// TIA Portal project "Project1" (V15)

(* hardware
DEVICE "PC-System_1"  SIMATIC PC station
   slot 0: "SIMATIC PC station"  Rail  SIMATIC PC-Station  V1.0
      slot 125: "Stationmanager"  Station_Manager  V6.0.4
   slot 1: "HMI_RT_1"  WinCC RT Professional  6AV2 105-0xxxx-xxxx  15.0.0.0
   slot 2: "IE general_1"  IE General  IE_CP  V8.2.0
DEVICE "S7-1200 station_1"  S7-1200 Station
   slot 0: "Rack_0"  S7-1200 Rack  Rack  V1.0
   slot 1: "PLC_1"  CPU 1212C DC/DC/DC  6ES7 212-1AE40-0XB0  V4.2
*)

// ===== PLC "PLC_1"  CPU 1212C DC/DC/DC =====

VAR_GLOBAL   // PLC tag table "Default tag table"
   "In1" AT %M0.0 : Bool;
   "Out1" AT %M0.1 : Bool;
END_VAR

ORGANIZATION_BLOCK "Main"   // OB1, LAD, ProgramCycle
TITLE = "Main Program Sweep (Cycle)"
{ S7_Optimized_Access := 'TRUE' }
VERSION : 0.1
   VAR_INPUT
      Initial_Call : Bool;   // Initial call of this OB
      Remanence : Bool;   // =True, if remanent data are available
   END_VAR
BEGIN

REGION Network 1
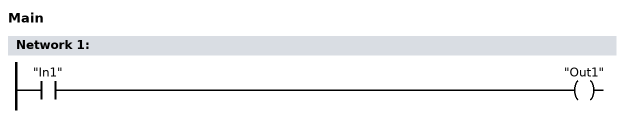
   RUNG wire#powerrail
      Contact( "In1" )
      Coil( "Out1" )
   END_RUNG
   // the same network as SCL:
   "Out1" := "In1";
END_REGION
END_ORGANIZATION_BLOCK

(* ===== HMI "HMI_RT_1" =====
system functions are stored by id; their names below are inferred from use
connection "S7-1200": S71200_TCP_IP, SCADA_S7_1200

HMI tags "Default tag table"
   "In1" : Bool = PLC In1 AT %M0.0, 500 ms
   "Out1" : Bool = PLC Out1 AT %M0.1, 500 ms

screen "Screen_1" 1024x768
   Button "Button_1" at 141,218 size 80x30; TextOff 'Go'
      on PressLeft: SetBit("In1")
      on ReleaseLeft: ResetBit("In1")
      Appearance <- "Out1"
*)